# EPICS autosave request: optics/opticsApp/Db/ASRPmirrorTable_settings.req
$(P)$(TBL):fixedPointZ
$(P)$(TBL):pitchArmLen
